// TwinCAT 3 PLC project SymbolTable
// ProgramVersion: 3.1.4022.6
// libraries:
//   Tc2_Standard, * (Beckhoff Automation GmbH)
//   Tc2_System, * (Beckhoff Automation GmbH)
//   Tc3_Module, * (Beckhoff Automation GmbH)
// project tree:
//   DUTs/ADS/ AdsDatatypeEntry.TcDUT (not stored), AdsSymbolEntry.TcDUT (not stored), AdsSymbolUploadInfo.TcDUT (not stored), AdsSymbolUploadInfo2.TcDUT
//   DUTs/ TReadSymbolTableState.TcDUT
//   GVLs/ GVL.TcGVL
//   / PlcTask.TcTTO
//   POUs/ AnalyseSymbolTable.TcPOU, LogMsg.TcPOU, MAIN.TcPOU
// real-time tasks:
//   TASK PlcTask: cycle T#1ms, priority 20, ADS port 351

CONFIGURATION SymbolTable
    RESOURCE PLC ON TwinCAT3
        TASK PlcTask(INTERVAL := T#1ms, PRIORITY := 20);
        PROGRAM MAIN WITH PlcTask : MAIN;
    END_RESOURCE
END_CONFIGURATION

// ---- DUTs/ADS/AdsSymbolUploadInfo2.TcDUT
TYPE AdsSymbolUploadInfo2 :
STRUCT
   nSymbols : UDINT;
   nSymSize : UDINT;
   nDatatypes : UDINT;
   nDatatypeSize : UDINT;
   nMaxDynSymbols : UDINT;
   nUsedDynSymbols : UDINT;
END_STRUCT
END_TYPE

// ---- DUTs/TReadSymbolTableState.TcDUT
{attribute 'to_string'}
TYPE TReadSymbolTableState :
(
	RS_WAIT_FOR_START,
	RS_READ_SYMBOL_UPLOAD_INFO,
	RS_READ_SYMBOL_UPLOAD,
	RS_PROCESS_SYMBOL_UPLOAD,
	
	RS_READ_SYMBOL_UPLOAD_INFO2,
	RS_READ_DATA_TYPE_UPLOAD,
	RS_PROCESS_DATA_UPLOAD,
	RS_DONE
	
);
END_TYPE

// ---- GVLs/GVL.TcGVL
VAR_GLOBAL
	gTime:	UDINT;
	gTraceNumber:	UDINT;
END_VAR

// ---- POUs/MAIN.TcPOU
PROGRAM MAIN
VAR
	AdsRead:						ADSREADEX;
	ADSReadWrite:					ADSRDWRT;
	SymbolUploadInfo:				AdsSymbolUploadInfo;
	DestBuffer:						ARRAY [0..100] OF BYTE;
	SrcBuffer:						STRING;
	pTypeInfo:						POINTER TO BYTE;
	ReadSymbolTableState:			TReadSymbolTableState;
	ReadSymbolTableStatePrev:		TReadSymbolTableState;
	StateEntry:						BOOL := TRUE;
	start:							BOOL;
	pAdsSymbolEntry:				POINTER TO AdsSymbolEntry;
	pSubAdsSymbolEntry:				POINTER TO AdsSymbolEntry;
	pNameStringPointer:				POINTER TO STRING;
	pTypeStringPointer:				POINTER TO STRING;
	pCommentStringPointer:			POINTER TO STRING;
	NameString:						STRING;
	TypeString:						STRING;
	CommentString:					STRING;
	pSubNameStringPointer:			POINTER TO STRING;
	SubNameString:					STRING;
	iterate:						BOOL;
	i:								UDINT;

	SymbolUploadInfo2:				AdsSymbolUploadInfo2;
	pDataInfo:						POINTER TO BYTE;
	pAdsDatatypeEntry:				POINTER TO AdsDatatypeEntry;
	pSubAdsDatatypeEntry:			POINTER TO AdsDatatypeEntry;
	AnalyseSymbolTable:				AnalyseSymbolTable;
	
	
END_VAR

CASE ReadSymbolTableState OF
	RS_WAIT_FOR_START:
		IF(start = TRUE)THEN 	
			start := FALSE;			
			ReadSymbolTableState := RS_READ_SYMBOL_UPLOAD_INFO;
		END_IF
		
	RS_READ_SYMBOL_UPLOAD_INFO:	
		
		AdsRead(PORT := 851, 
				DESTADDR := ADR(SymbolUploadInfo),
				IDXGRP := 16#F00C,
				IDXOFFS := 0,
				LEN := SIZEOF(SymbolUploadInfo),
				READ := TRUE
				);
		IF(AdsRead.BUSY = FALSE)THEN
			AdsRead(Read := FALSE);
			pTypeInfo := __NEW(BYTE, SymbolUploadInfo.nSymSize);			
			ReadSymbolTableState := RS_READ_SYMBOL_UPLOAD;	
		END_IF	
		
	RS_READ_SYMBOL_UPLOAD: 			
		AdsRead(PORT := 851, 
				DESTADDR := pTypeInfo,
				IDXGRP := 16#F00B,
				IDXOFFS := 0,
				LEN := SymbolUploadInfo.nSymSize,
				READ := TRUE
				);
		IF(AdsRead.BUSY = FALSE)THEN
			AdsRead(Read := FALSE);						
			ReadSymbolTableState := RS_PROCESS_SYMBOL_UPLOAD;		
		END_IF
			
	RS_PROCESS_SYMBOL_UPLOAD:
		IF(StateEntry)THEN
			i := 0;
			pAdsSymbolEntry := pTypeInfo;
		END_IF
		IF(i< SymbolUploadInfo.nSymbols-1)THEN
			pNameStringPointer := pAdsSymbolEntry + 30 (* Sizeof(AdsDatatypeEntry) geeft net wat teveel*);
			NameString := pNameStringPointer^;
			//LogMsg(NameString);
			
 			pTypeStringPointer := pNameStringPointer + pAdsSymbolEntry^.nameLength + 1;
			TypeString := pTypeStringPointer^;
			
			pCommentStringPointer := pTypeStringPointer + pAdsSymbolEntry^.typeLength + 1;
			CommentString := pCommentStringPointer^;
			
			LogMsg(concat(concat(concat(concat(NameString,' '), TypeString), ' '), CommentString));
	
			pAdsSymbolEntry := pAdsSymbolEntry + pAdsSymbolEntry^.entryLength;
			i := i + 1;
		ELSE
			ReadSymbolTableState := RS_READ_SYMBOL_UPLOAD_INFO2;
		END_IF
		

	RS_READ_SYMBOL_UPLOAD_INFO2:
		AdsRead(
			PORT := 851, 
			DESTADDR := ADR(SymbolUploadInfo2),
			IDXGRP := 16#F00F,
			IDXOFFS := 0,
			LEN := SIZEOF(SymbolUploadInfo2),
			READ := TRUE);
			
		IF(AdsRead.BUSY = FALSE)THEN
			AdsRead(Read := FALSE);
			pDataInfo := __NEW(BYTE, SymbolUploadInfo2.nDatatypeSize);			
			ReadSymbolTableState := RS_READ_DATA_TYPE_UPLOAD;	
		END_IF	
		
		
	RS_READ_DATA_TYPE_UPLOAD:
		AdsRead(
				PORT := 851, 
				DESTADDR := pDataInfo,
				IDXGRP := 16#F00E,
				IDXOFFS := 0,
				LEN := SymbolUploadInfo2.nDatatypeSize,
				READ := TRUE);

		IF(AdsRead.BUSY = FALSE)THEN			
			ReadSymbolTableState := RS_PROCESS_DATA_UPLOAD;
		END_IF
		
	RS_PROCESS_DATA_UPLOAD:
		IF(StateEntry)THEN
			i := 0;
			pAdsDatatypeEntry := pDataInfo;
		END_IF
		IF (i < SymbolUploadInfo2.nDatatypes-1) THEN
				
			AnalyseSymbolTable.AnalyseAdsDatatpe(pAdsDatatypeEntry, '');			
			
			i := i + 1;
			pAdsDatatypeEntry := pAdsDatatypeEntry + pAdsDatatypeEntry^.entryLength;
		ELSE
			ReadSymbolTableState := RS_DONE;
		END_IF
		
	RS_DONE:
		;		

100:
	ADSReadWrite(
		PORT := 851,
		SRCADDR :=  ADR(SrcBuffer),
		DESTADDR := ADR(DestBuffer)
			);
END_CASE
(*
CASE ReadSymbolTableState OF
	0:
		IF(start = TRUE)THEN 	
			start := FALSE;
			AdsRead(
				PORT := 851, 
				DESTADDR := ADR(SymbolUploadInfo),
				IDXGRP := 16#F00F,
				IDXOFFS := 0,
				LEN := SIZEOF(SymbolUploadInfo),
				READ := TRUE
					);
			ReadSymbolTableState := 1;
		END_IF
		
	1:	
		AdsRead();
		IF(AdsRead.BUSY = FALSE)THEN
			AdsRead(Read := FALSE);
			pTypeInfo := __NEW(BYTE, SymbolUploadInfo.nDatatypeSize);			
			ReadSymbolTableState := 2;	
		END_IF	
		
	2:
		AdsRead();
		IF(AdsRead.BUSY = FALSE)THEN
			AdsRead(
				PORT := 851, 
				DESTADDR := pTypeInfo,
				IDXGRP := 16#F00E,
				IDXOFFS := 0,
				LEN := SymbolUploadInfo.nDatatypeSize,
				READ := TRUE
					);
			ReadSymbolTableState := 3;
		END_IF
		
	3: 		
		AdsRead();
		IF(AdsRead.BUSY = FALSE)THEN
			pAdsDatatypeEntry := pTypeInfo;
			ReadSymbolTableState := 4;
		END_IF
			
	4:
		FOR i := 0 TO SymbolUploadInfo.nDatatypes DO
					
			pNameStringPointer := pAdsDatatypeEntry + 42 (* Sizeof(AdsDatatypeEntry) geeft net wat teveel*);
			NameString := pNameStringPointer^;
			TracePrintString(NameString);
			IF(NameString = 'TSymbolUploadInfo')THEN
				iterate := FALSE;	
			END_IF
			IF(pAdsDatatypeEntry^.subItems > 0)THEN
				//Sub item:
				pSubAdsDatatypeEntry := pNameStringPointer + pAdsDatatypeEntry^.nameLength+1 + pAdsDatatypeEntry^.typeLength+1 + pAdsDatatypeEntry^.commentLength+1 + 8; 
				pSubNameStringPointer := pSubAdsDatatypeEntry + 42 (* Sizeof(AdsDatatypeEntry) geeft net wat teveel*);
				SubNameString := pSubNameStringPointer^;
				TracePrintString(SubNameString);
			END_IF			
			pAdsDatatypeEntry := pAdsDatatypeEntry + pAdsDatatypeEntry^.entryLength;
		END_FOR
		ReadSymbolTableState := 5;
		
		

100:
	ADSReadWrite(
		PORT := 851,
		SRCADDR :=  ADR(SrcBuffer),
		DESTADDR := ADR(DestBuffer)
			);
END_CASE

*)

LogStateChange();

gTime := gTime + 1;

METHOD LogStateChange : BOOL
VAR_INPUT
END_VAR
IF(ReadSymbolTableState <> ReadSymbolTableStatePrev)THEN
	LogMsg(concat(concat(TO_STRING(ReadSymbolTableStatePrev), ' => '), TO_STRING(ReadSymbolTableState)));
	StateEntry := TRUE;
ELSE
	StateEntry := FALSE;
END_IF
ReadSymbolTableStatePrev := ReadSymbolTableState;
END_METHOD

END_PROGRAM

// ---- POUs/AnalyseSymbolTable.TcPOU
FUNCTION_BLOCK AnalyseSymbolTable
VAR_INPUT
END_VAR
VAR_OUTPUT
END_VAR
VAR
END_VAR

{attribute 'estimated-stack-usage' := 100000}
METHOD AnalyseAdsDatatpe : BOOL
VAR_INPUT
	pAdsDatatypeEntry:	POINTER TO AdsDatatypeEntry;
	PrependString:		STRING;
END_VAR
VAR
	pSubAdsDatatypeEntry:			POINTER TO AdsDatatypeEntry;
	pNameStringPointer:				POINTER TO STRING;
	pTypeStringPointer:				POINTER TO STRING;
	pCommentStringPointer:			POINTER TO STRING;
	NameString:						STRING;
	TypeString:						STRING;
	CommentString:					STRING;
	i:								UDINT;
END_VAR
pNameStringPointer := pAdsDatatypeEntry + 42 (* Sizeof(AdsDatatypeEntry) geeft net wat teveel*);
NameString := pNameStringPointer^;
//LogMsg(NameString);

pTypeStringPointer := pNameStringPointer + pAdsDatatypeEntry^.nameLength + 1;
TypeString := pTypeStringPointer^;

pCommentStringPointer := pTypeStringPointer + pAdsDatatypeEntry^.typeLength + 1;
CommentString := pCommentStringPointer^;

pSubAdsDatatypeEntry := pCommentStringPointer + pAdsDatatypeEntry^.commentLength + 1;

pSubAdsDatatypeEntry := pSubAdsDatatypeEntry + pAdsDatatypeEntry^.arrayDim * 16;

LogMsg(concat(concat(concat(concat(concat(PrependString, NameString),' '), TypeString), ' '), CommentString));

IF(pAdsDatatypeEntry^.arrayDim > 0)THEN
	LogMsg(concat(concat(PrependString,'Array dimension: '), TO_STRING(pAdsDatatypeEntry^.arrayDim)));
END_IF	

IF(pAdsDatatypeEntry^.subItems > 0)THEN
	//Sub item:
	LogMsg(concat(concat(PrependString,'Amount of Subitems: '), TO_STRING(pAdsDatatypeEntry^.subItems)));
	FOR i := 0 TO pAdsDatatypeEntry^.subItems-1 DO
		THIS^.AnalyseAdsDatatpe(pSubAdsDatatypeEntry, '  ');
		pSubAdsDatatypeEntry := pSubAdsDatatypeEntry + pSubAdsDatatypeEntry^.entryLength;
	END_FOR

END_IF
END_METHOD

END_FUNCTION_BLOCK

// ---- POUs/LogMsg.TcPOU
FUNCTION LogMsg : DINT
VAR_INPUT
	aString:	STRING;
END_VAR
VAR
	gSubTimeStr:	STRING;
END_VAR

LogMsg := ADSLOGSTR( ADSLOG_MSGTYPE_HINT OR ADSLOG_MSGTYPE_LOG, 'PLC: %s', concat(concat(concat(concat(UDINT_TO_STRING(gTraceNumber),': '), UDINT_TO_STRING(gTime)), ': '), aString));
gTraceNumber := gTraceNumber + 1;

END_FUNCTION
